// Mitsubishi GX Works2 project: dmddyd1   PLC: Q02/Q02H

PROGRAM MAIN
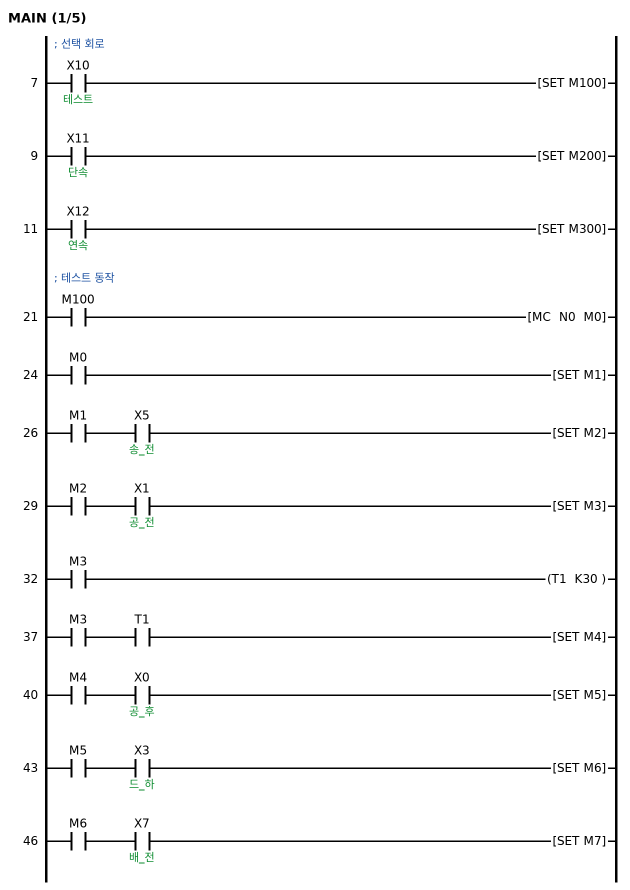
; 선택 회로
7     LD      X10  ; 테스트
      SET     M100
9     LD      X11  ; 단속
      SET     M200
11    LD      X12  ; 연속
      SET     M300
; 테스트 동작
21    LD      M100
      MC      N0 M0
24    LD      M0
      SET     M1
26    LD      M1
      AND     X5  ; 송_전
      SET     M2
29    LD      M2
      AND     X1  ; 공_전
      SET     M3
32    LD      M3
      OUT     T1 K30
37    LD      M3
      AND     T1
      SET     M4
40    LD      M4
      AND     X0  ; 공_후
      SET     M5
43    LD      M5
      AND     X3  ; 드_하
      SET     M6
46    LD      M6
      AND     X7  ; 배_전
      SET     M7
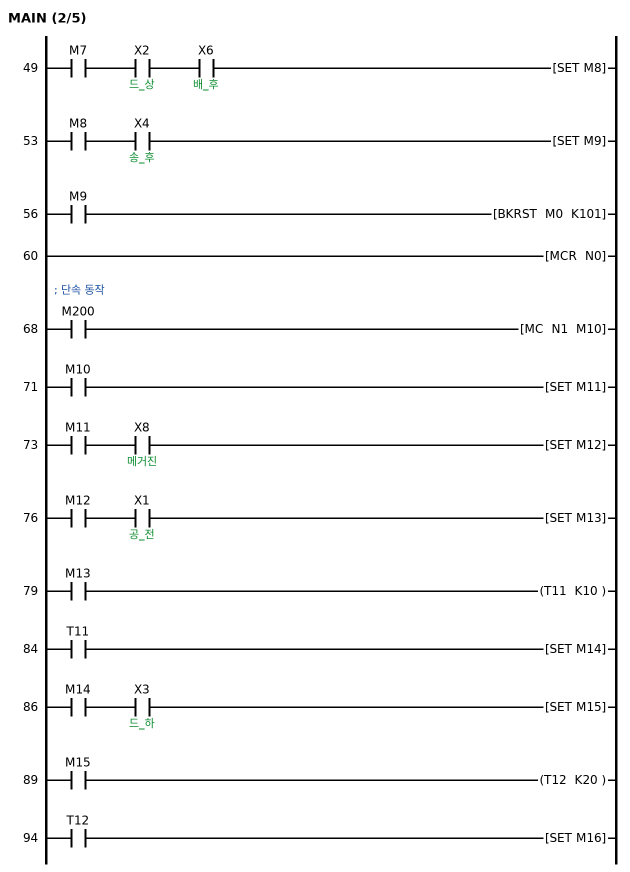
49    LD      M7
      AND     X2  ; 드_상
      AND     X6  ; 배_후
      SET     M8
53    LD      M8
      AND     X4  ; 송_후
      SET     M9
56    LD      M9
      BKRST   M0 K101
60    MCR     N0
; 단속 동작
68    LD      M200
      MC      N1 M10
71    LD      M10
      SET     M11
73    LD      M11
      AND     X8  ; 메거진
      SET     M12
76    LD      M12
      AND     X1  ; 공_전
      SET     M13
79    LD      M13
      OUT     T11 K10
84    LD      T11
      SET     M14
86    LD      M14
      AND     X3  ; 드_하
      SET     M15
89    LD      M15
      OUT     T12 K20
94    LD      T12
      SET     M16
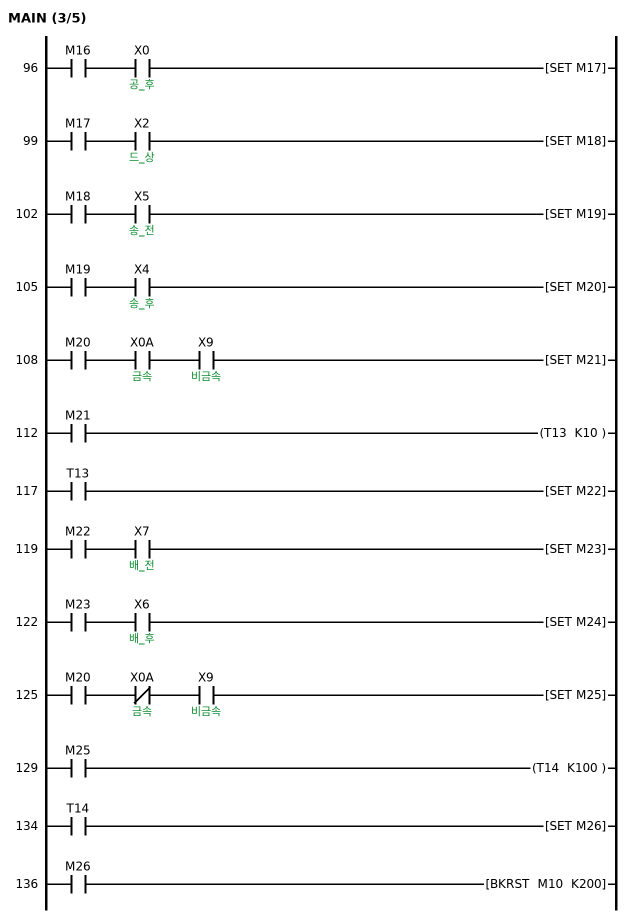
96    LD      M16
      AND     X0  ; 공_후
      SET     M17
99    LD      M17
      AND     X2  ; 드_상
      SET     M18
102   LD      M18
      AND     X5  ; 송_전
      SET     M19
105   LD      M19
      AND     X4  ; 송_후
      SET     M20
108   LD      M20
      AND     X0A  ; 금속
      AND     X9  ; 비금속
      SET     M21
112   LD      M21
      OUT     T13 K10
117   LD      T13
      SET     M22
119   LD      M22
      AND     X7  ; 배_전
      SET     M23
122   LD      M23
      AND     X6  ; 배_후
      SET     M24
125   LD      M20
      ANI     X0A  ; 금속
      AND     X9  ; 비금속
      SET     M25
129   LD      M25
      OUT     T14 K100
134   LD      T14
      SET     M26
136   LD      M26
      BKRST   M10 K200
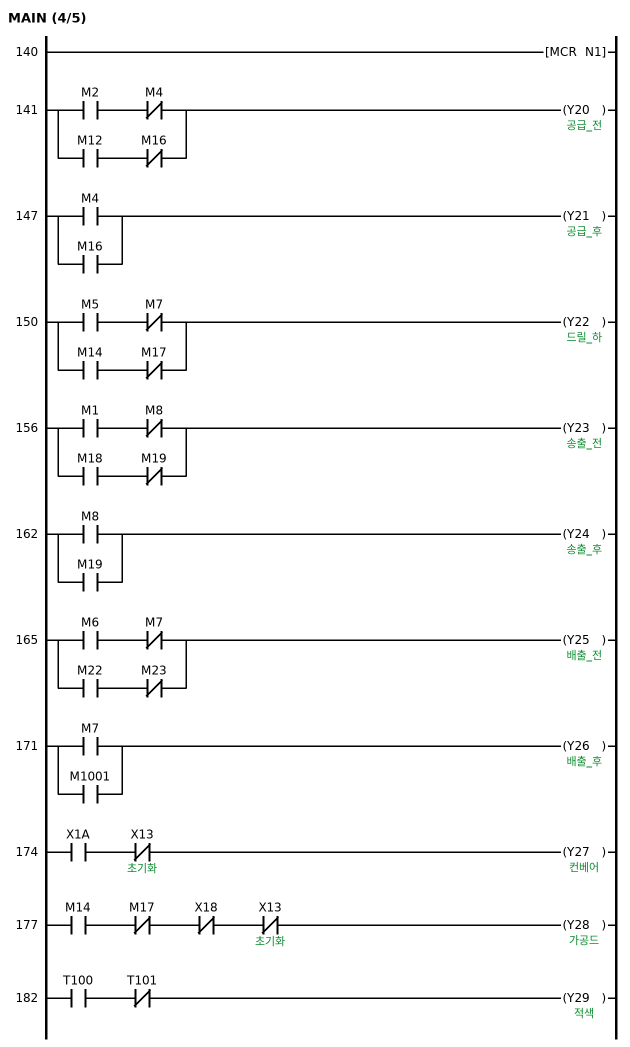
140   MCR     N1
141   LD      M2
      ANI     M4
      LD      M12
      ANI     M16
      ORB
      OUT     Y20  ; 공급_전
147   LD      M4
      OR      M16
      OUT     Y21  ; 공급_후
150   LD      M5
      ANI     M7
      LD      M14
      ANI     M17
      ORB
      OUT     Y22  ; 드릴_하
156   LD      M1
      ANI     M8
      LD      M18
      ANI     M19
      ORB
      OUT     Y23  ; 송출_전
162   LD      M8
      OR      M19
      OUT     Y24  ; 송출_후
165   LD      M6
      ANI     M7
      LD      M22
      ANI     M23
      ORB
      OUT     Y25  ; 배출_전
171   LD      M7
      OR      M1001
      OUT     Y26  ; 배출_후
174   LD      X1A
      ANI     X13  ; 초기화
      OUT     Y27  ; 컨베어
177   LD      M14
      ANI     M17
      ANI     X18
      ANI     X13  ; 초기화
      OUT     Y28  ; 가공드
182   LD      T100
      ANI     T101
      OUT     Y29  ; 적색
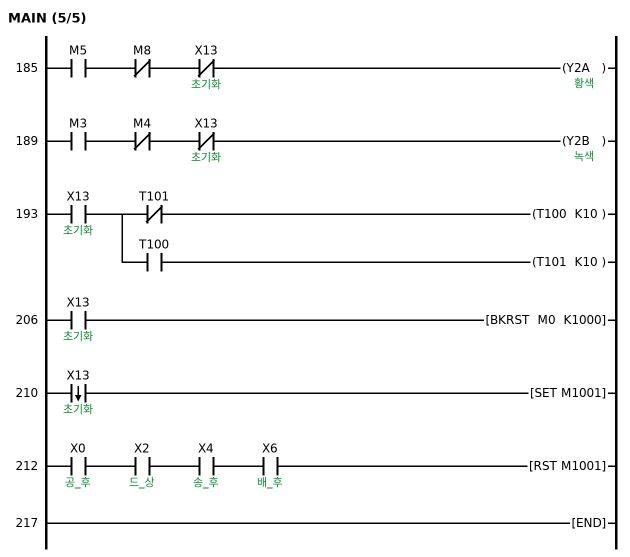
185   LD      M5
      ANI     M8
      ANI     X13  ; 초기화
      OUT     Y2A  ; 황색
189   LD      M3
      ANI     M4
      ANI     X13  ; 초기화
      OUT     Y2B  ; 녹색
193   LD      X13  ; 초기화
      MPS
      ANI     T101
      OUT     T100 K10
      MPP
      AND     T100
      OUT     T101 K10
206   LD      X13  ; 초기화
      BKRST   M0 K1000
210   LDF     X13  ; 초기화
      SET     M1001
212   LD      X0  ; 공_후
      AND     X2  ; 드_상
      AND     X4  ; 송_후
      AND     X6  ; 배_후
      RST     M1001
217   END
END_PROGRAM

PROGRAM MAIN1
0     END
END_PROGRAM
